TEXTLIST TextList_SettingPage
  1 = '1'
  2 = '2'
  3 = '3'
  4 = '4'
  5 = '5'
  6 = '6'
  7 = 'LOADING'
  8 = 'UNLOADING'
  9 = 'GENERAL'
   = ''
END_TEXTLIST

(* stored: Version 1.1.0.1, ProductVersion 3.1.4024.12
   TextList TextList_SettingPage: Id {e3bfcec1-903e-46cb-8238-a6bb24c91890} *)
